{attribute 'qualified_only'}
VAR_GLOBAL CONSTANT
    ADDRESS     : STRING := '13 Apple Cart Way'; // Next door to 1 Pear Drop Lane
    N_BEDROOMS  : USINT  := 4;
    N_BATHROOMS : USINT  := 1;
END_VAR

(* stored: Version 1.1.0.1, ProductVersion 3.1.4024.13
   GVL house: Id {53cf6feb-0caa-459b-8425-8ca72f64350e} *)
